FUNCTION_BLOCK TRDC
  (* Standard: 61499-2 *)
  (* Version 0.1, 2015-00-16, Th?o, PC_THEO *)
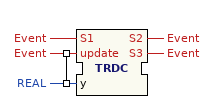
  EVENT_INPUT
    S1;
    update WITH y;
  END_EVENT
  EVENT_OUTPUT
    S2;
    S3;
  END_EVENT
  VAR_INPUT
    y : REAL;
  END_VAR
  VAR
    ice_id : INT;
  END_VAR
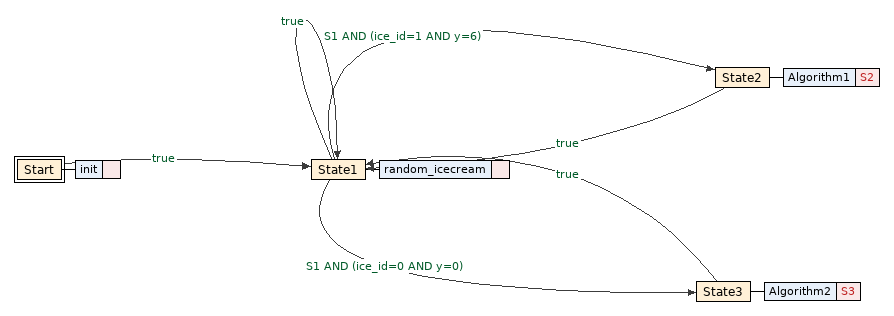
  EC_STATES
    Start : init;
    State1 : random_icecream;
    State2 : Algorithm1 -> S2;
    State3 : Algorithm2 -> S3;
  END_STATES
  EC_TRANSITIONS
    Start TO State1 := true;
    State1 TO State2 := S1 AND (ice_id=1 AND y=6);
    State1 TO State3 := S1 AND (ice_id=0 AND y=0);
    State1 TO State1 := true;
    State2 TO State1 := true;
    State3 TO State1 := true;
  END_TRANSITIONS
  ALGORITHM init IN C:
me->ice_id=2;
  END_ALGORITHM
  ALGORITHM random_icecream IN C:
/* Intializes random number generator */
srand(time(NULL));

me->ice_id = rand() % 2 ;

//printf("%d, %f\n", me->ice_id, me->y);
  END_ALGORITHM
  ALGORITHM Algorithm1 IN C:
//printf("S2\n");
printf("Send signal: divert to the storage1\n");
  END_ALGORITHM
  ALGORITHM Algorithm2 IN C:
//printf("S3\n");
printf("Send signal: divert to the storage2\n");
  END_ALGORITHM
END_FUNCTION_BLOCK
